// LS Electric XG5000 project: Automated Warehouse
// PLC LSPLC

PROGRAM AutomatedWarehouse (task: 스캔 프로그램)

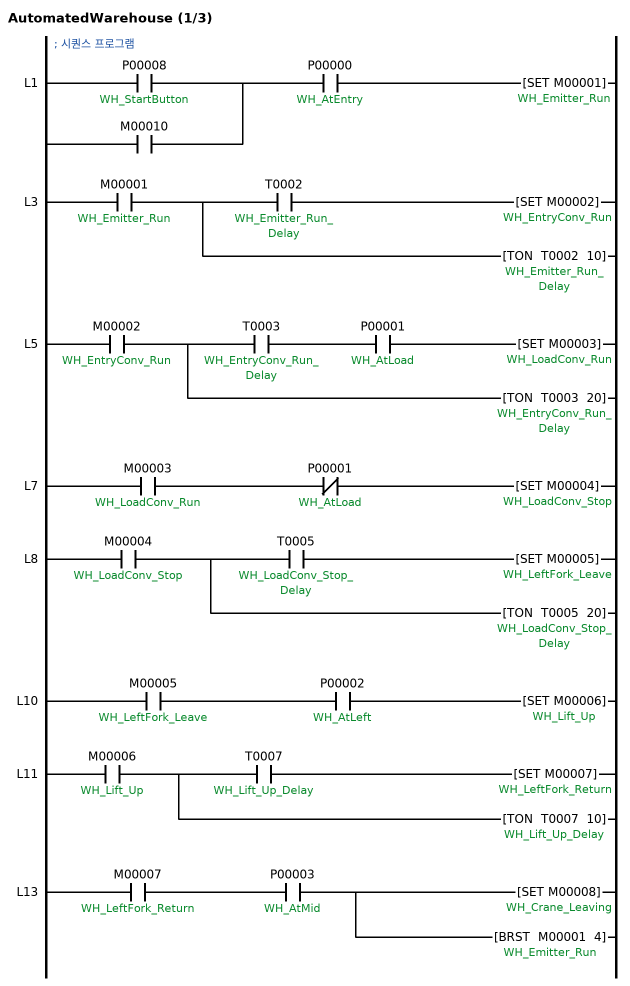
// 시퀀스 프로그램
; L1
LOAD      P00008	// WH_StartButton
OR        M00010
AND       P00000	// WH_AtEntry
SET       M00001	// WH_Emitter_Run
; L3
LOAD      M00001	// WH_Emitter_Run
MPUSH
AND       T0002	// WH_Emitter_Run_Delay
SET       M00002	// WH_EntryConv_Run
MPOP
TON       T0002 10	// WH_Emitter_Run_Delay
; L5
LOAD      M00002	// WH_EntryConv_Run
MPUSH
AND       T0003	// WH_EntryConv_Run_Delay
AND       P00001	// WH_AtLoad
SET       M00003	// WH_LoadConv_Run
MPOP
TON       T0003 20	// WH_EntryConv_Run_Delay
; L7
LOAD      M00003	// WH_LoadConv_Run
AND NOT   P00001	// WH_AtLoad
SET       M00004	// WH_LoadConv_Stop
; L8
LOAD      M00004	// WH_LoadConv_Stop
MPUSH
AND       T0005	// WH_LoadConv_Stop_Delay
SET       M00005	// WH_LeftFork_Leave
MPOP
TON       T0005 20	// WH_LoadConv_Stop_Delay
; L10
LOAD      M00005	// WH_LeftFork_Leave
AND       P00002	// WH_AtLeft
SET       M00006	// WH_Lift_Up
; L11
LOAD      M00006	// WH_Lift_Up
MPUSH
AND       T0007	// WH_Lift_Up_Delay
SET       M00007	// WH_LeftFork_Return
MPOP
TON       T0007 10	// WH_Lift_Up_Delay
; L13
LOAD      M00007	// WH_LeftFork_Return
AND       P00003	// WH_AtMid
SET       M00008	// WH_Crane_Leaving
BRST      M00001 4	// WH_Emitter_Run

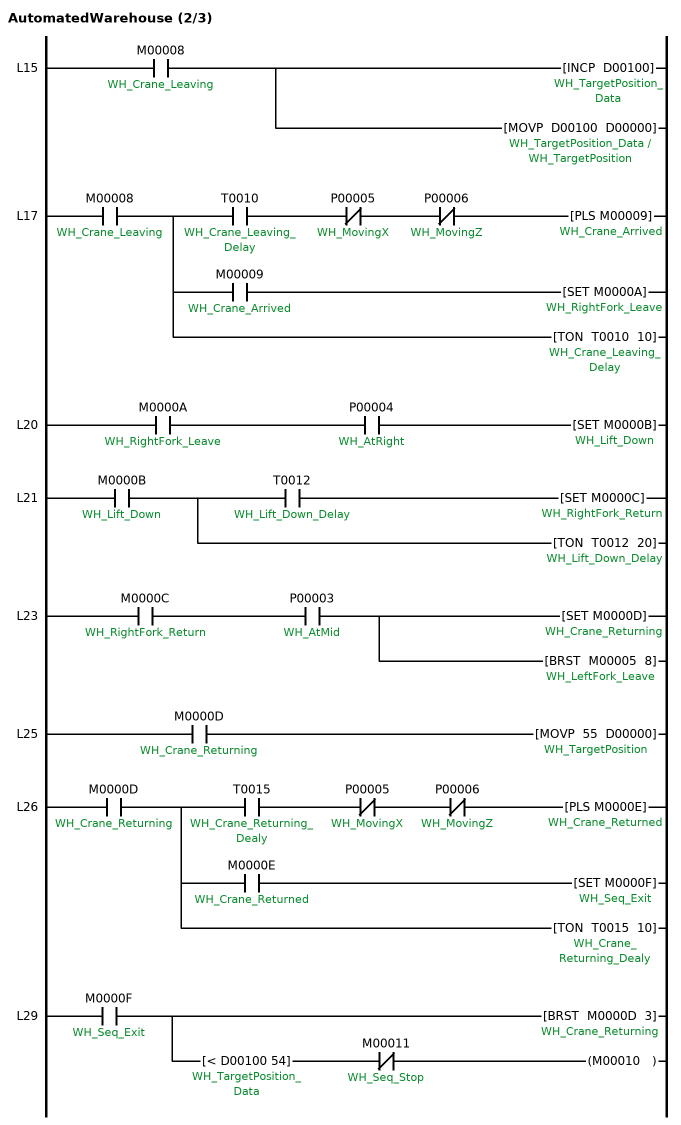
; L15
LOAD      M00008	// WH_Crane_Leaving
INCP      D00100	// WH_TargetPosition_Data
MOVP      D00100 D00000	// WH_TargetPosition_Data / WH_TargetPosition
; L17
LOAD      M00008	// WH_Crane_Leaving
MPUSH
AND       T0010	// WH_Crane_Leaving_Delay
AND NOT   P00005	// WH_MovingX
AND NOT   P00006	// WH_MovingZ
OUTP      M00009	// WH_Crane_Arrived
MLOAD
AND       M00009	// WH_Crane_Arrived
SET       M0000A	// WH_RightFork_Leave
MPOP
TON       T0010 10	// WH_Crane_Leaving_Delay
; L20
LOAD      M0000A	// WH_RightFork_Leave
AND       P00004	// WH_AtRight
SET       M0000B	// WH_Lift_Down
; L21
LOAD      M0000B	// WH_Lift_Down
MPUSH
AND       T0012	// WH_Lift_Down_Delay
SET       M0000C	// WH_RightFork_Return
MPOP
TON       T0012 20	// WH_Lift_Down_Delay
; L23
LOAD      M0000C	// WH_RightFork_Return
AND       P00003	// WH_AtMid
SET       M0000D	// WH_Crane_Returning
BRST      M00005 8	// WH_LeftFork_Leave
; L25
LOAD      M0000D	// WH_Crane_Returning
MOVP      55 D00000	// WH_TargetPosition
; L26
LOAD      M0000D	// WH_Crane_Returning
MPUSH
AND       T0015	// WH_Crane_Returning_Dealy
AND NOT   P00005	// WH_MovingX
AND NOT   P00006	// WH_MovingZ
OUTP      M0000E	// WH_Crane_Returned
MLOAD
AND       M0000E	// WH_Crane_Returned
SET       M0000F	// WH_Seq_Exit
MPOP
TON       T0015 10	// WH_Crane_Returning_Dealy
; L29
LOAD      M0000F	// WH_Seq_Exit
BRST      M0000D 3	// WH_Crane_Returning
AND<      D00100 54	// WH_TargetPosition_Data
AND NOT   M00011	// WH_Seq_Stop
OUT       M00010

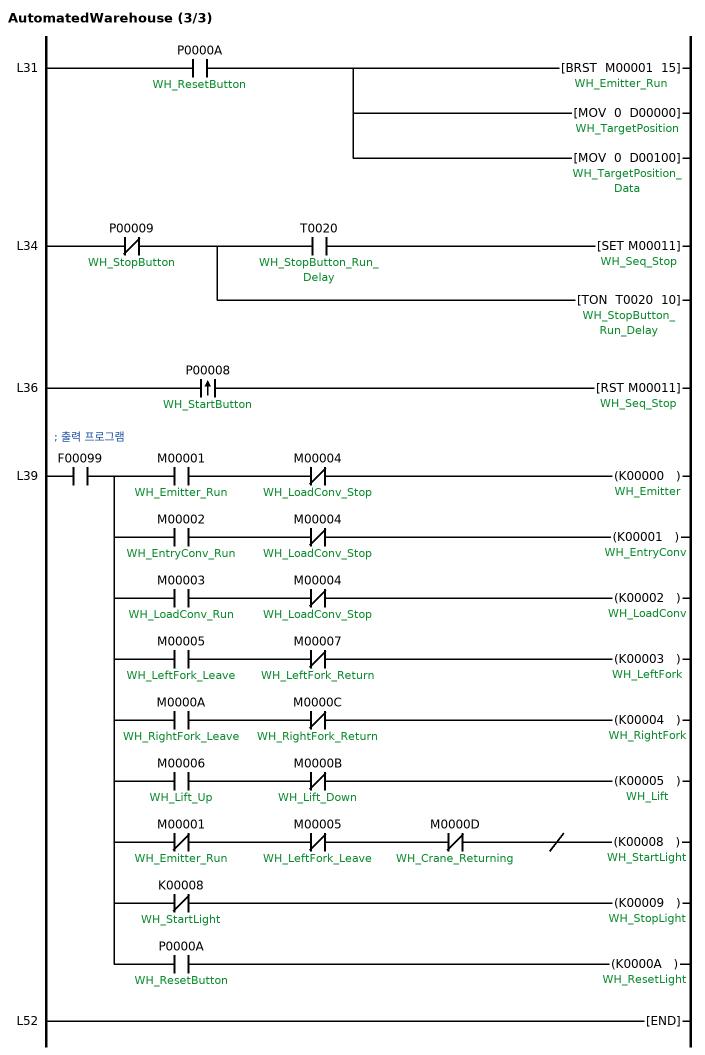
; L31
LOAD      P0000A	// WH_ResetButton
BRST      M00001 15	// WH_Emitter_Run
MOV       0 D00000	// WH_TargetPosition
MOV       0 D00100	// WH_TargetPosition_Data
; L34
LOAD NOT  P00009	// WH_StopButton
MPUSH
AND       T0020	// WH_StopButton_Run_Delay
SET       M00011	// WH_Seq_Stop
MPOP
TON       T0020 10	// WH_StopButton_Run_Delay
; L36
LOADP     P00008	// WH_StartButton
RST       M00011	// WH_Seq_Stop
// 출력 프로그램
; L39
LOAD      F00099
MPUSH
AND       M00001	// WH_Emitter_Run
AND NOT   M00004	// WH_LoadConv_Stop
OUT       K00000	// WH_Emitter
MLOAD
AND       M00002	// WH_EntryConv_Run
AND NOT   M00004	// WH_LoadConv_Stop
OUT       K00001	// WH_EntryConv
MLOAD
AND       M00003	// WH_LoadConv_Run
AND NOT   M00004	// WH_LoadConv_Stop
OUT       K00002	// WH_LoadConv
MLOAD
AND       M00005	// WH_LeftFork_Leave
AND NOT   M00007	// WH_LeftFork_Return
OUT       K00003	// WH_LeftFork
MLOAD
AND       M0000A	// WH_RightFork_Leave
AND NOT   M0000C	// WH_RightFork_Return
OUT       K00004	// WH_RightFork
MLOAD
AND       M00006	// WH_Lift_Up
AND NOT   M0000B	// WH_Lift_Down
OUT       K00005	// WH_Lift
MLOAD
AND NOT   M00001	// WH_Emitter_Run
AND NOT   M00005	// WH_LeftFork_Leave
AND NOT   M0000D	// WH_Crane_Returning
NOT
OUT       K00008	// WH_StartLight
MLOAD
AND NOT   K00008	// WH_StartLight
OUT       K00009	// WH_StopLight
MPOP
AND       P0000A	// WH_ResetButton
OUT       K0000A	// WH_ResetLight
; L52
END